FUNCTION_BLOCK SlaveCylinder_TEST (* Basic Function Block Type *)
  (* Standard: 61499-2 *)
  (* Version 0.2, 2003-12-04, JHC, Rockwell Automation, Renamed for better indexing. *)
  (* Version 0.1, 2002-11-05, JHC, Rockwell Automation, Corrected missing ST element in Algorithm REQ. *)
  (* Version 0.0, 2000-05-30, JHC, Rockwell Automation *)
  (* Compiler header: package fb.rt.pnp; *)
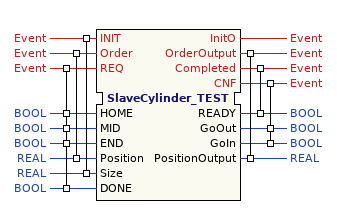
  EVENT_INPUT
    INIT WITH Size;
    Order WITH Position;
    REQ WITH HOME, MID, END, DONE;
  END_EVENT
  EVENT_OUTPUT
    InitO;
    OrderOutput WITH PositionOutput;
    Completed WITH READY; (* Initialization Confirm *)
    CNF WITH GoOut, GoIn;
  END_EVENT
  VAR_INPUT
    HOME : BOOL; (* Input event qualifier *)
    MID : BOOL; (* Input event qualifier *)
    END : BOOL; (* Input event qualifier *)
    Position : REAL;
    Size : REAL;
    DONE : BOOL;
  END_VAR
  VAR_OUTPUT
    READY : BOOL; (* Output event qualifier *)
    GoOut : BOOL; (* Output event qualifier *)
    GoIn : BOOL; (* Output event qualifier *)
    PositionOutput : REAL;
  END_VAR
  VAR
    init : BOOL;
    extended : BOOL;
    GoCenter : BOOL;
    PositionO : REAL;
  END_VAR
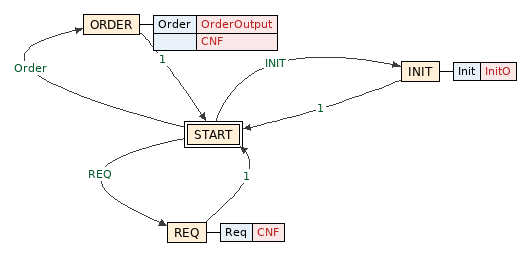
  EC_STATES
    START; (* Initial State *)
    ORDER : Order -> OrderOutput, -> CNF; (* Initialization *)
    REQ : Req -> CNF; (* Normal execution *)
    INIT : Init -> InitO;
  END_STATES
  EC_TRANSITIONS
    START TO ORDER := Order;
    START TO REQ := REQ;
    ORDER TO START := 1;
    REQ TO START := 1;
    START TO INIT := INIT;
    INIT TO START := 1;
  END_TRANSITIONS
  ALGORITHM Init IN Java: (* Initialization algorithm *)
if(!init.value) {
init.value = true;
GoOut.value=false;
GoIn.value=false;
GoCenter.value=false;
READY.value=true;
extended.value=false;
}
System.out.println("initcyl!!!");
  END_ALGORITHM
  ALGORITHM Order IN Java: (* Initialization algorithm *)
READY.value=false;
GoOut.value=false;
GoCenter.value=false;
GoIn.value=false;

if(Position.value >= Size.value) {
GoOut.value=true;
PositionO.value = Position.value - Size.value;
} else {
if(Position.value == 1 && Size.value == 2) {
GoCenter.value=true;
GoIn.value=true;
PositionO.value = Position.value - 1;
} else {
GoIn.value=true;
PositionO.value = Position.value;
}

}





PositionOutput.value = PositionO.value;
  END_ALGORITHM
  ALGORITHM Req IN Java: (* Initialization algorithm *)
if(HOME.value && GoIn.value) {
GoOut.value=false;
GoIn.value=false;
extended.value=false;
}

if(END.value && GoOut.value) {
GoOut.value=false;
GoIn.value=false;
extended.value=true;
}

if(END.value && GoCenter.value) {
GoOut.value=false;
GoIn.value=true;
extended.value=false;
}
if(HOME.value && GoCenter.value) {
GoOut.value=true;
GoIn.value=false;
extended.value=false;
}
if(MID.value && GoCenter.value) {
GoOut.value=false;
GoIn.value=false;
extended.value=false;
}

if(!GoOut.value && !GoIn.value && DONE.value) {
READY.value=true;
}
if(Size.value == 2 && MID.value) {
System.out.println("Req:"+MID.value);
}
  END_ALGORITHM
END_FUNCTION_BLOCK
